# EPICS autosave request: iocBoot/ioc2Pumps/auto_settings.req
file "ISCOController_settings.req" P=$(P)
file "ISCOPumpN_settings.req",     P=$(P), PUMP=A:
file "ISCOPumpN_settings.req",     P=$(P), PUMP=B:
